(* Logix 5000 project; controller cow Emulate 5570 rev 36.11; software revision 36.00; part 6 of 6 *)
(* tags used below, declared in another part *)
   Batch_delay : TIMER;
   Big_Add : TIMER;
   Big_Avg : REAL;
   Big_Bin_Changed : BOOL;
   Big_Bridge_time : TIMER;
   Big_Error_Over : BOOL;
   Big_ErrorWeight : REAL;
   Big_id : DINT;
   Big_id1 : DINT;
   Big_Idx : DINT;
   Big_Index : DINT;
   Big_Run_Fs : BOOL;
   Big_Scale1 : REAL;
   Big_Scale2 : REAL;
   Big_Scale3 : REAL;
   Big_Timer : TIMER;
   BigBin_Change_ID : DINT;
   Bin_Index : DINT;
   Find : BOOL;
   Hand_Index : DINT;
   Hand_Scale1 : REAL;
   Index : DINT;
   INDEX1 : DINT;
   Max_BigID : DINT;
   No_Big_CMD : BOOL;
   Ons : BOOL[64];
   Part_Index : DINT;
   rcp_Big1 : Part_Type;
   rcp_Big_Bridge_delay : TIMER;
   rcp_BigBin_Bridge : DINT;
   rcp_BigLastID1 : DINT;
   Recipe_Mult : CONTROL;
   Report_TIMER : TIMER;
   Scale_Simulate_Timer : TIMER;
   Simulate_Big_w : REAL;
   ZERO : DINT[100];
   Bin01 : ALIAS FOR rcp_Big_Bin[0];
   Bin02 : ALIAS FOR rcp_Big_Bin[1];
   Bin03 : ALIAS FOR rcp_Big_Bin[2];
   Bin04 : ALIAS FOR rcp_Big_Bin[3];
   Bin05 : ALIAS FOR rcp_Big_Bin[4];
   Bin06 : ALIAS FOR rcp_Big_Bin[5];
   Bin07 : ALIAS FOR rcp_Big_Bin[6];
   Bin08 : ALIAS FOR rcp_Big_Bin[7];
   Bin09 : ALIAS FOR rcp_Big_Bin[8];
   Bin10 : ALIAS FOR rcp_Big_Bin[9];
   Bin11 : ALIAS FOR rcp_Big_Bin[10];
   Bin12 : ALIAS FOR rcp_Big_Bin[11];
   Bin13 : ALIAS FOR rcp_Big_Bin[12];
   Bin14 : ALIAS FOR rcp_Big_Bin[13];
   Bin15 : ALIAS FOR rcp_Big_Bin[14];
   Bin16 : ALIAS FOR rcp_Big_Bin[15];
   E331 : SCALE_WEIGHT;
   E351 : Valve;
   E352 : Valve;
   LED_Batch_seq : DINT;
   LED_Batch_Total : ALIAS FOR rcp_Recipe.BatchSet;
   Led_Hand_PartNumber : DINT;
   Led_Hand_RealWeight : REAL;
   LED_Hand_SetWeight : REAL;
   Now : DateTime_Type;
   rcp_Auto : ALIAS FOR SYS_E.AUTO;
   rcp_Batch : DINT;
   rcp_Batch_OK : BOOL;
   rcp_Batch_Start : BOOL;
   rcp_Big : Part_Type;
   rcp_Big_Add : BOOL;
   rcp_Big_Add_Cmd : BOOL;
   rcp_Big_Add_Skip : BOOL;
   rcp_Big_Bin : Bin_Raw[20];
   rcp_Big_Bridge : BOOL;
   rcp_Big_Bridge_skip : BOOL;
   rcp_Big_Continue : BOOL;
   rcp_Big_Pause : BOOL;
   rcp_Big_Run : BOOL;
   rcp_Big_Scale : REAL;
   rcp_Big_Speed : DINT;
   rcp_BigBin_Change : DINT;
   rcp_BigLastID : DINT;
   rcp_Cancel_Pause : BOOL;
   rcp_class : DINT;
   rcp_Clear : BOOL;
   rcp_Dest_Bin : DINT;
   rcp_Hand : Part_Type_Hand;
   rcp_Hand_Index : DINT;
   rcp_Hand_PB : BOOL;
   rcp_Hand_Run : BOOL;
   rcp_Hand_Scale : REAL;
   rcp_Hand_Total : DINT;
   rcp_Mult : REAL;
   rcp_Recipe : Recipe_Type;
   rcp_Recipe_pNumber : DINT[20];
   rcp_Recipe_Power_Reset : BOOL;
   rcp_Recipe_pSetweight : REAL[20];
   rcp_Recipe_Reset : BOOL;
   rcp_Report_Bin : INT[66];
   rcp_Report_Log : BOOL;
   rcp_Report_Number : DINT[60];
   rcp_Report_RealWeight : REAL[60];
   rcp_Report_SetWeight : REAL[60];
   rcp_RUN : BOOL;
   rcp_Scale_Lock : BOOL;
   rcp_schedule : Recipe_Type[11];
   rcp_schedule_Index : DINT;
   rcp_Schedule_INPUT : BOOL;
   rcp_ScheduleLog : ScheduleLog[10];
   rcp_Set_Pause : BOOL;
   SCALE_SIMULATE : BOOL;
   SYS : System_Common;
(* Recipe, continued *)

ROUTINE MainRoutine   (* ladder *)
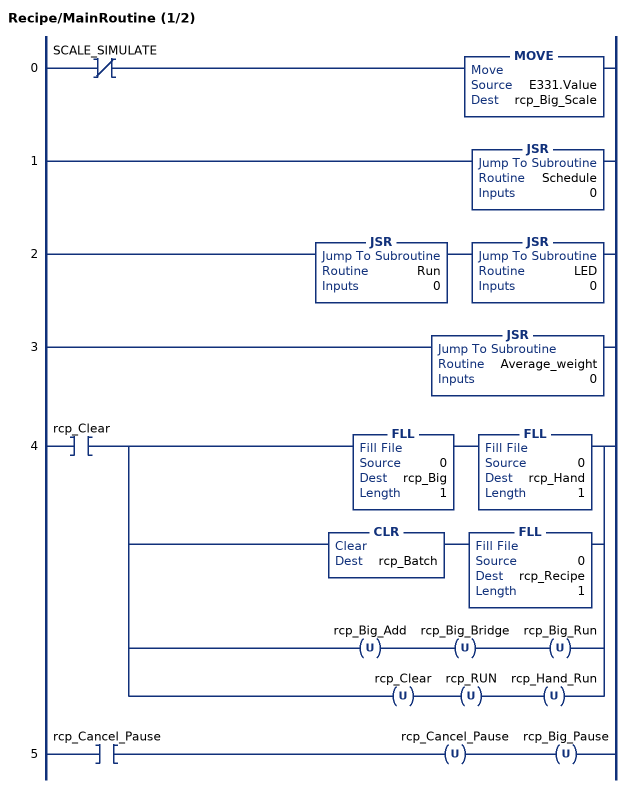
   0: XIO(SCALE_SIMULATE)MOVE(E331.Value,rcp_Big_Scale);
   1: JSR(Schedule,0);
   2: JSR(Run,0)JSR(LED,0);
   3: JSR(Average_weight,0);
   4: XIC(rcp_Clear)[FLL(0,rcp_Big,1) FLL(0,rcp_Hand,1) ,CLR(rcp_Batch) FLL(0,rcp_Recipe,1) ,OTU(rcp_Big_Add) OTU(rcp_Big_Bridge) OTU(rcp_Big_Run) ,OTU(rcp_Clear) OTU(rcp_RUN) OTU(rcp_Hand_Run) ];
   5: XIC(rcp_Cancel_Pause)OTU(rcp_Cancel_Pause)OTU(rcp_Big_Pause);
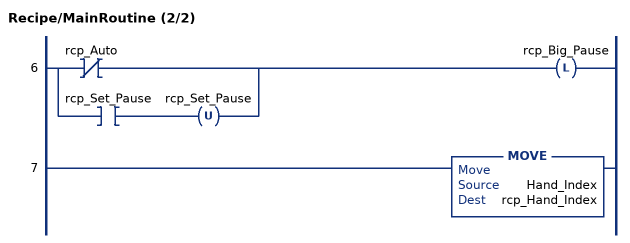
   6: [XIO(rcp_Auto) ,XIC(rcp_Set_Pause) OTU(rcp_Set_Pause) ]OTL(rcp_Big_Pause);
   7: MOVE(Hand_Index,rcp_Hand_Index);
END_ROUTINE

ROUTINE Run   (* ladder *)
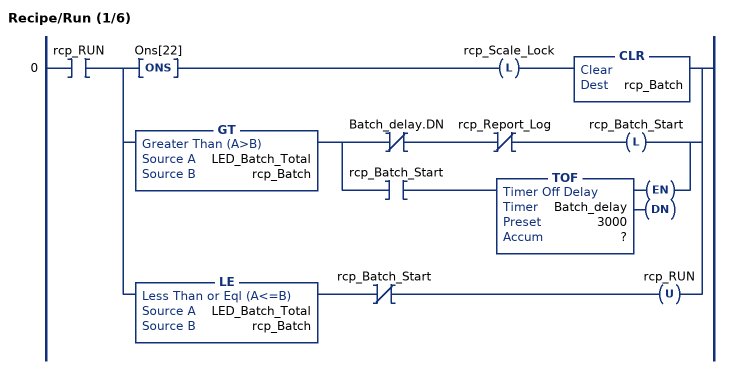
   0: XIC(rcp_RUN)[ONS(Ons[22]) OTL(rcp_Scale_Lock) CLR(rcp_Batch) ,GT(LED_Batch_Total,rcp_Batch) [XIO(Batch_delay.DN) XIO(rcp_Report_Log) OTL(rcp_Batch_Start) ,XIC(rcp_Batch_Start) TOF(Batch_delay,?,?) ] ,LE(LED_Batch_Total,rcp_Batch) XIO(rcp_Batch_Start) OTU(rcp_RUN) ];
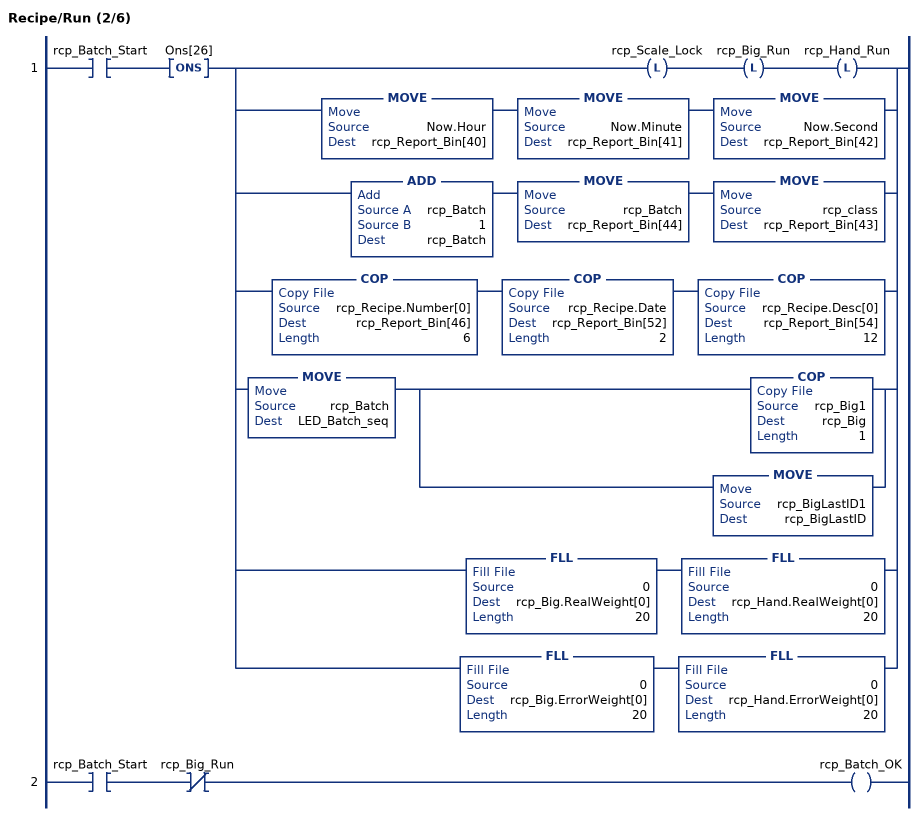
   1: XIC(rcp_Batch_Start)ONS(Ons[26])[OTL(rcp_Scale_Lock) OTL(rcp_Big_Run) OTL(rcp_Hand_Run) ,MOVE(Now.Hour,rcp_Report_Bin[40]) MOVE(Now.Minute,rcp_Report_Bin[41]) MOVE(Now.Second,rcp_Report_Bin[42]) ,ADD(rcp_Batch,1,rcp_Batch) MOVE(rcp_Batch,rcp_Report_Bin[44]) MOVE(rcp_class,rcp_Report_Bin[43]) ,COP(rcp_Recipe.Number[0],rcp_Report_Bin[46],6) COP(rcp_Recipe.Date,rcp_Report_Bin[52],2) COP(rcp_Recipe.Desc[0],rcp_Report_Bin[54],12) ,MOVE(rcp_Batch,LED_Batch_seq) [COP(rcp_Big1,rcp_Big,1) ,MOVE(rcp_BigLastID1,rcp_BigLastID) ] ,FLL(0,rcp_Big.RealWeight[0],20) FLL(0,rcp_Hand.RealWeight[0],20) ,FLL(0,rcp_Big.ErrorWeight[0],20) FLL(0,rcp_Hand.ErrorWeight[0],20) ];
   2: XIC(rcp_Batch_Start)XIO(rcp_Big_Run)OTE(rcp_Batch_OK);
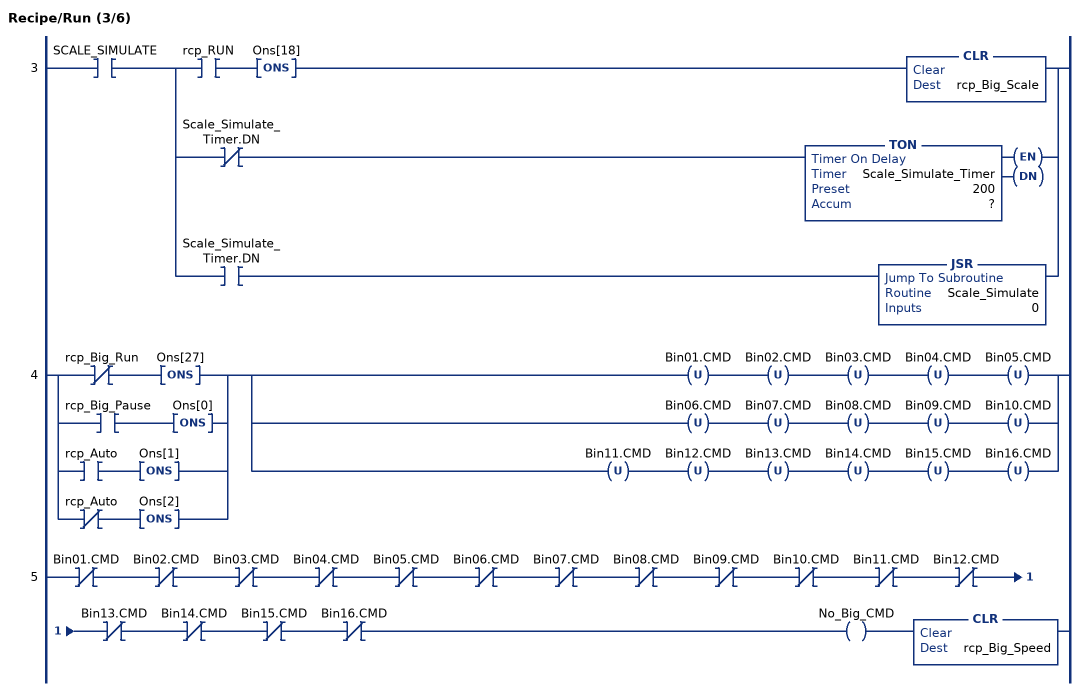
   3: XIC(SCALE_SIMULATE)[XIC(rcp_RUN) ONS(Ons[18]) CLR(rcp_Big_Scale) ,XIO(Scale_Simulate_Timer.DN) TON(Scale_Simulate_Timer,?,?) ,XIC(Scale_Simulate_Timer.DN) JSR(Scale_Simulate,0) ];
   4: [XIO(rcp_Big_Run) ONS(Ons[27]) ,XIC(rcp_Big_Pause) ONS(Ons[0]) ,XIC(rcp_Auto) ONS(Ons[1]) ,XIO(rcp_Auto) ONS(Ons[2]) ][OTU(Bin01.CMD) OTU(Bin02.CMD) OTU(Bin03.CMD) OTU(Bin04.CMD) OTU(Bin05.CMD) ,OTU(Bin06.CMD) OTU(Bin07.CMD) OTU(Bin08.CMD) OTU(Bin09.CMD) OTU(Bin10.CMD) ,OTU(Bin11.CMD) OTU(Bin12.CMD) OTU(Bin13.CMD) OTU(Bin14.CMD) OTU(Bin15.CMD) OTU(Bin16.CMD) ];
   5: XIO(Bin01.CMD)XIO(Bin02.CMD)XIO(Bin03.CMD)XIO(Bin04.CMD)XIO(Bin05.CMD)XIO(Bin06.CMD)XIO(Bin07.CMD)XIO(Bin08.CMD)XIO(Bin09.CMD)XIO(Bin10.CMD)XIO(Bin11.CMD)XIO(Bin12.CMD)XIO(Bin13.CMD)XIO(Bin14.CMD)XIO(Bin15.CMD)XIO(Bin16.CMD)OTE(No_Big_CMD)CLR(rcp_Big_Speed);
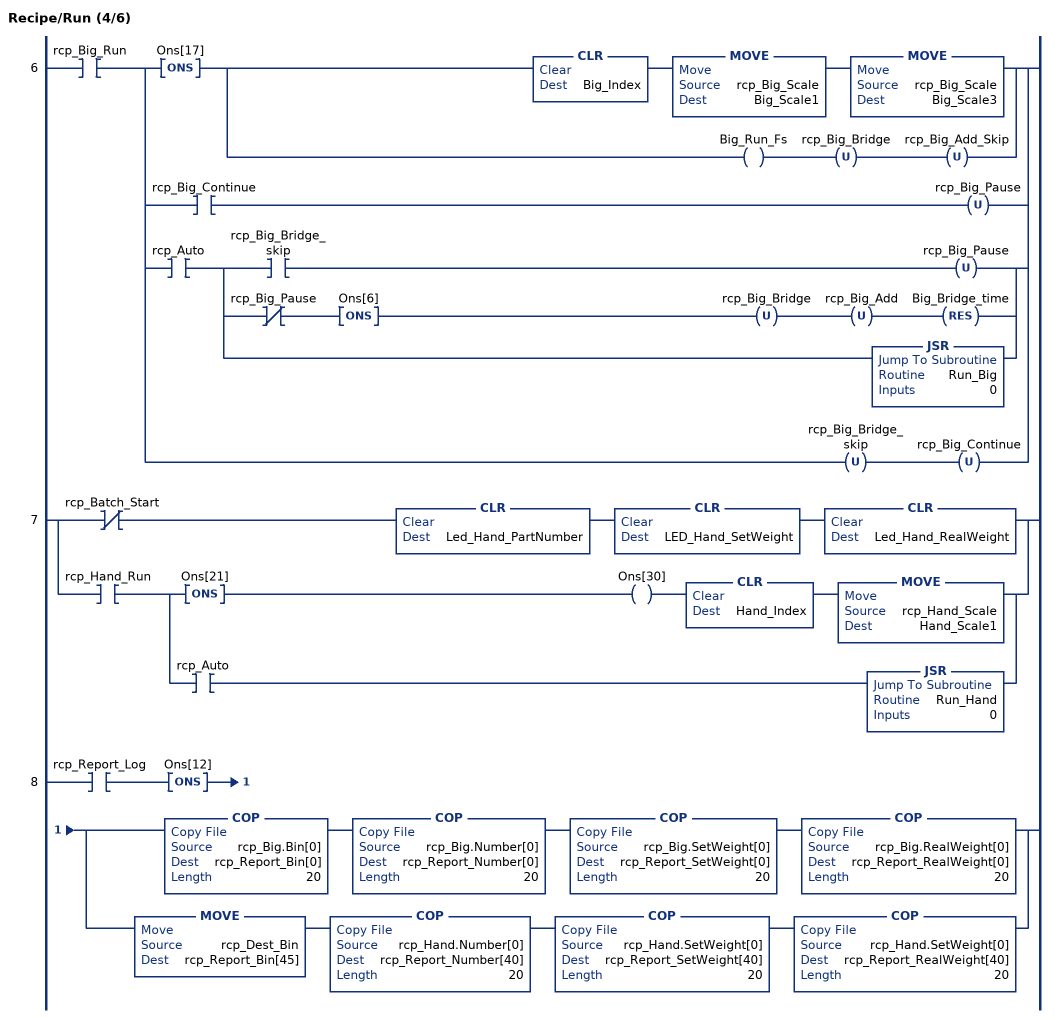
   6: XIC(rcp_Big_Run)[ONS(Ons[17]) [CLR(Big_Index) MOVE(rcp_Big_Scale,Big_Scale1) MOVE(rcp_Big_Scale,Big_Scale3) ,OTE(Big_Run_Fs) OTU(rcp_Big_Bridge) OTU(rcp_Big_Add_Skip) ] ,XIC(rcp_Big_Continue) OTU(rcp_Big_Pause) ,XIC(rcp_Auto) [XIC(rcp_Big_Bridge_skip) OTU(rcp_Big_Pause) ,[XIO(rcp_Big_Pause) ONS(Ons[6]) OTU(rcp_Big_Bridge) OTU(rcp_Big_Add) RES(Big_Bridge_time) ,JSR(Run_Big,0) ] ] ,OTU(rcp_Big_Bridge_skip) OTU(rcp_Big_Continue) ];
   7: [XIO(rcp_Batch_Start) CLR(Led_Hand_PartNumber) CLR(LED_Hand_SetWeight) CLR(Led_Hand_RealWeight) ,XIC(rcp_Hand_Run) [ONS(Ons[21]) OTE(Ons[30]) CLR(Hand_Index) MOVE(rcp_Hand_Scale,Hand_Scale1) ,XIC(rcp_Auto) JSR(Run_Hand,0) ] ];
   8: XIC(rcp_Report_Log)ONS(Ons[12])[COP(rcp_Big.Bin[0],rcp_Report_Bin[0],20) COP(rcp_Big.Number[0],rcp_Report_Number[0],20) COP(rcp_Big.SetWeight[0],rcp_Report_SetWeight[0],20) COP(rcp_Big.RealWeight[0],rcp_Report_RealWeight[0],20) ,MOVE(rcp_Dest_Bin,rcp_Report_Bin[45]) COP(rcp_Hand.Number[0],rcp_Report_Number[40],20) COP(rcp_Hand.SetWeight[0],rcp_Report_SetWeight[40],20) COP(rcp_Hand.SetWeight[0],rcp_Report_RealWeight[40],20) ];
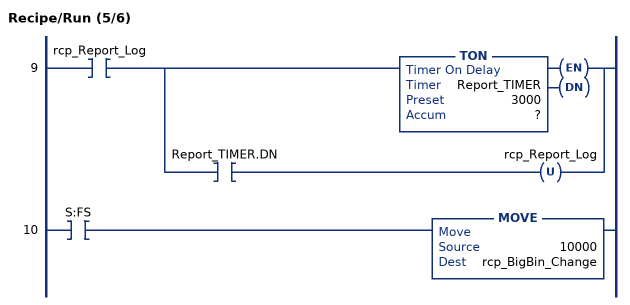
   9: XIC(rcp_Report_Log)[TON(Report_TIMER,?,?) ,XIC(Report_TIMER.DN) OTU(rcp_Report_Log) ];
   10: XIC(S:FS)MOVE(10000,rcp_BigBin_Change);
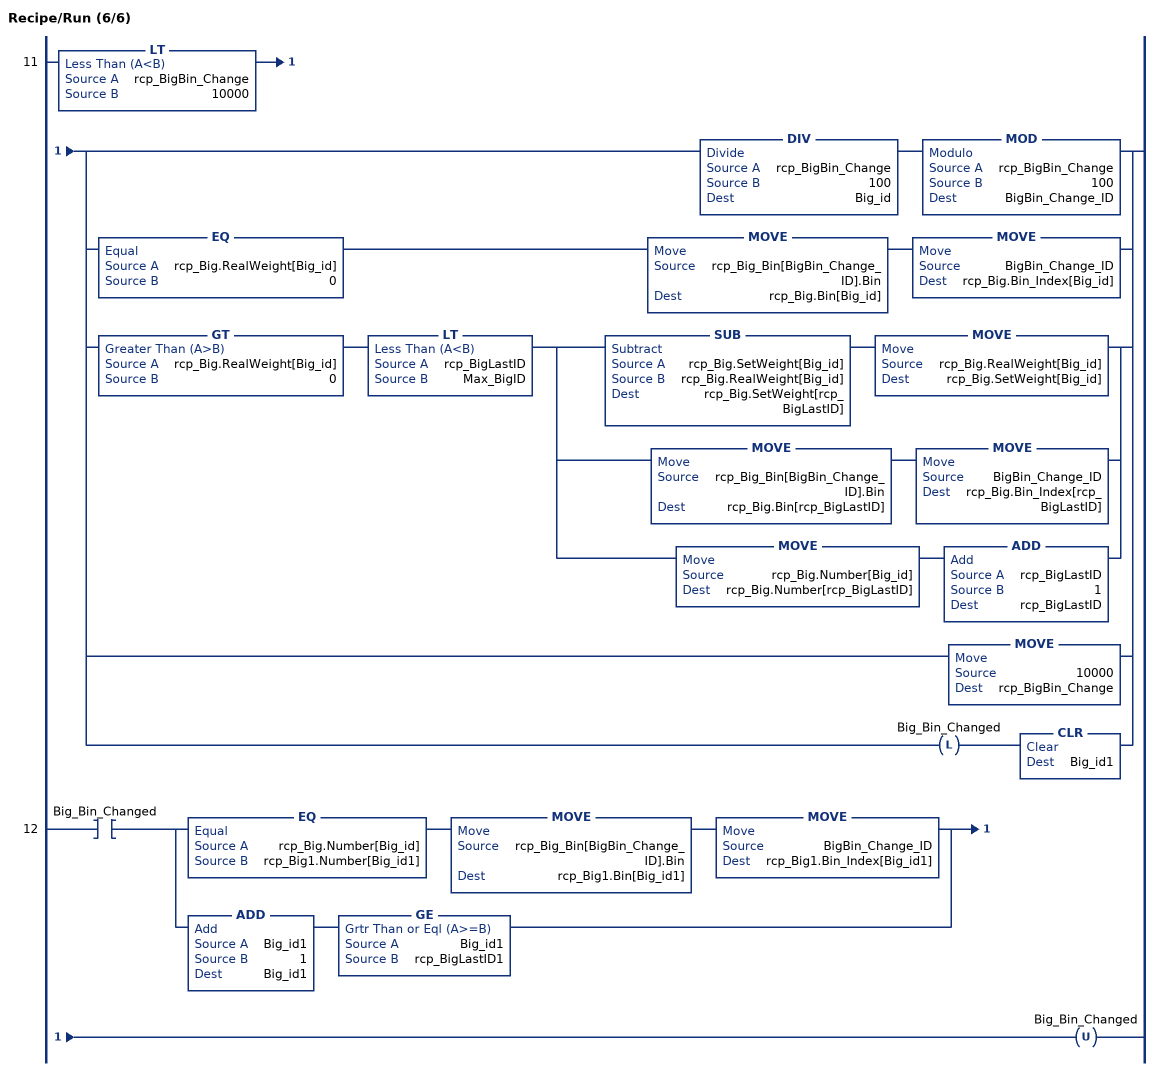
   11: LT(rcp_BigBin_Change,10000)[DIV(rcp_BigBin_Change,100,Big_id) MOD(rcp_BigBin_Change,100,BigBin_Change_ID) ,EQ(rcp_Big.RealWeight[Big_id],0) MOVE(rcp_Big_Bin[BigBin_Change_ID].Bin,rcp_Big.Bin[Big_id]) MOVE(BigBin_Change_ID,rcp_Big.Bin_Index[Big_id]) ,GT(rcp_Big.RealWeight[Big_id],0) LT(rcp_BigLastID,Max_BigID) [SUB(rcp_Big.SetWeight[Big_id],rcp_Big.RealWeight[Big_id],rcp_Big.SetWeight[rcp_BigLastID]) MOVE(rcp_Big.RealWeight[Big_id],rcp_Big.SetWeight[Big_id]) ,MOVE(rcp_Big_Bin[BigBin_Change_ID].Bin,rcp_Big.Bin[rcp_BigLastID]) MOVE(BigBin_Change_ID,rcp_Big.Bin_Index[rcp_BigLastID]) ,MOVE(rcp_Big.Number[Big_id],rcp_Big.Number[rcp_BigLastID]) ADD(rcp_BigLastID,1,rcp_BigLastID) ] ,MOVE(10000,rcp_BigBin_Change) ,OTL(Big_Bin_Changed) CLR(Big_id1) ];
   12: XIC(Big_Bin_Changed)[EQ(rcp_Big.Number[Big_id],rcp_Big1.Number[Big_id1]) MOVE(rcp_Big_Bin[BigBin_Change_ID].Bin,rcp_Big1.Bin[Big_id1]) MOVE(BigBin_Change_ID,rcp_Big1.Bin_Index[Big_id1]) ,ADD(Big_id1,1,Big_id1) GE(Big_id1,rcp_BigLastID1) ]OTU(Big_Bin_Changed);
END_ROUTINE

ROUTINE Run_Big   (* ladder *)
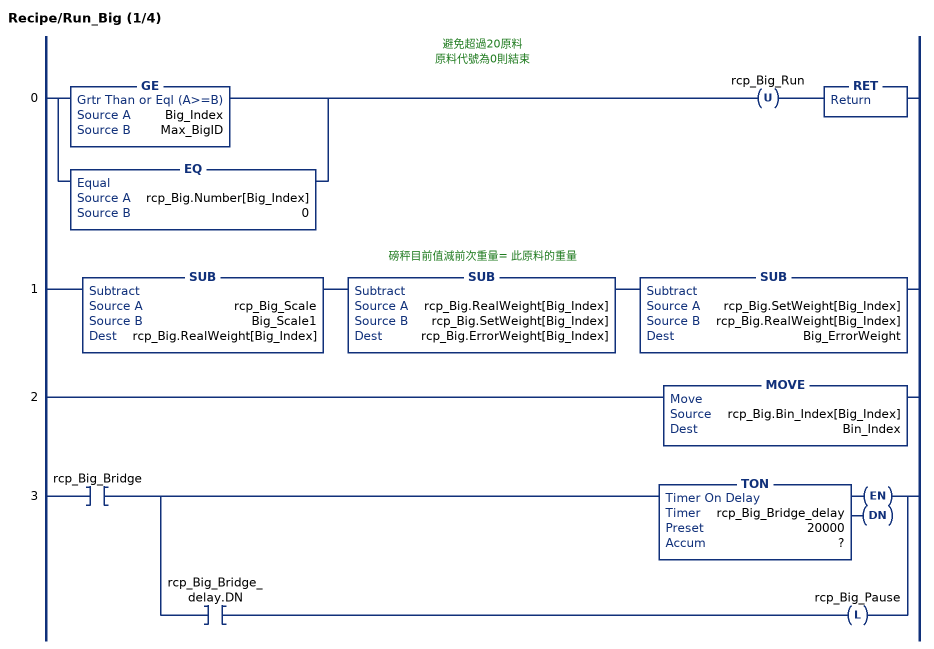
   // 避免超過20原料
   // 原料代號為0則結束
   0: [GE(Big_Index,Max_BigID) ,EQ(rcp_Big.Number[Big_Index],0) ]OTU(rcp_Big_Run)RET();
   // 磅秤目前值減前次重量= 此原料的重量
   1: SUB(rcp_Big_Scale,Big_Scale1,rcp_Big.RealWeight[Big_Index])SUB(rcp_Big.RealWeight[Big_Index],rcp_Big.SetWeight[Big_Index],rcp_Big.ErrorWeight[Big_Index])SUB(rcp_Big.SetWeight[Big_Index],rcp_Big.RealWeight[Big_Index],Big_ErrorWeight);
   2: MOVE(rcp_Big.Bin_Index[Big_Index],Bin_Index);
   3: XIC(rcp_Big_Bridge)[TON(rcp_Big_Bridge_delay,?,?) ,XIC(rcp_Big_Bridge_delay.DN) OTL(rcp_Big_Pause) ];
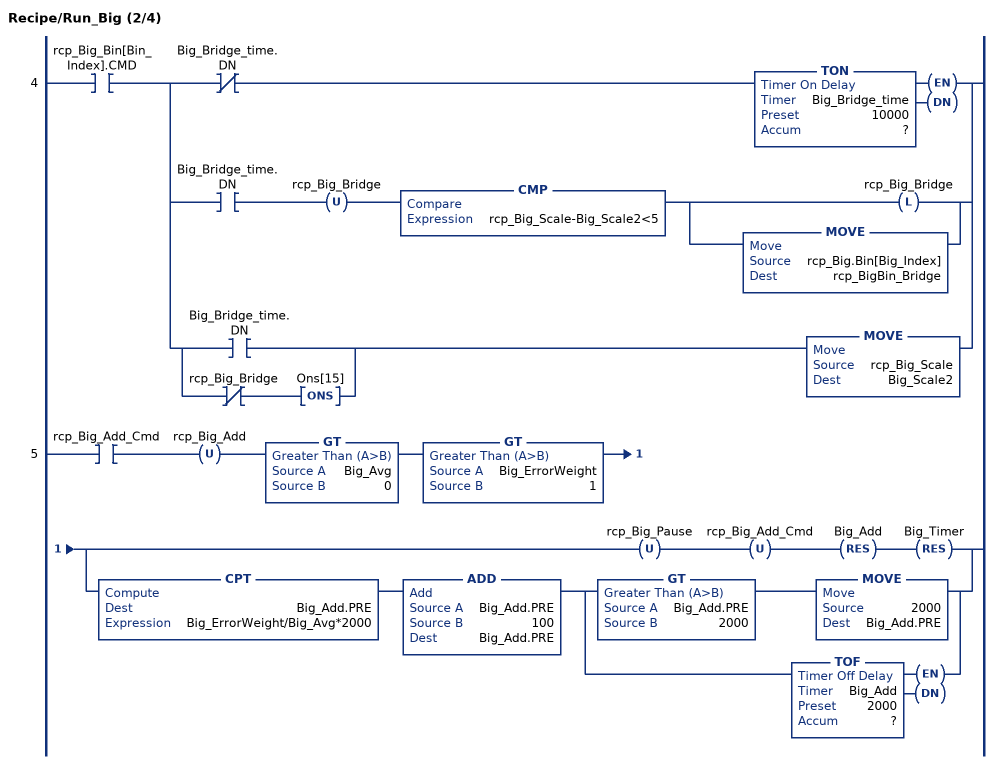
   4: XIC(rcp_Big_Bin[Bin_Index].CMD)[XIO(Big_Bridge_time.DN) TON(Big_Bridge_time,?,?) ,XIC(Big_Bridge_time.DN) OTU(rcp_Big_Bridge) CMP(rcp_Big_Scale-Big_Scale2<5) [OTL(rcp_Big_Bridge) ,MOVE(rcp_Big.Bin[Big_Index],rcp_BigBin_Bridge) ] ,[XIC(Big_Bridge_time.DN) ,XIO(rcp_Big_Bridge) ONS(Ons[15]) ] MOVE(rcp_Big_Scale,Big_Scale2) ];
   5: XIC(rcp_Big_Add_Cmd)OTU(rcp_Big_Add)GT(Big_Avg,0)GT(Big_ErrorWeight,1)[OTU(rcp_Big_Pause) OTU(rcp_Big_Add_Cmd) RES(Big_Add) RES(Big_Timer) ,CPT(Big_Add.PRE,Big_ErrorWeight/Big_Avg*2000) ADD(Big_Add.PRE,100,Big_Add.PRE) [GT(Big_Add.PRE,2000) MOVE(2000,Big_Add.PRE) ,TOF(Big_Add,?,?) ] ];
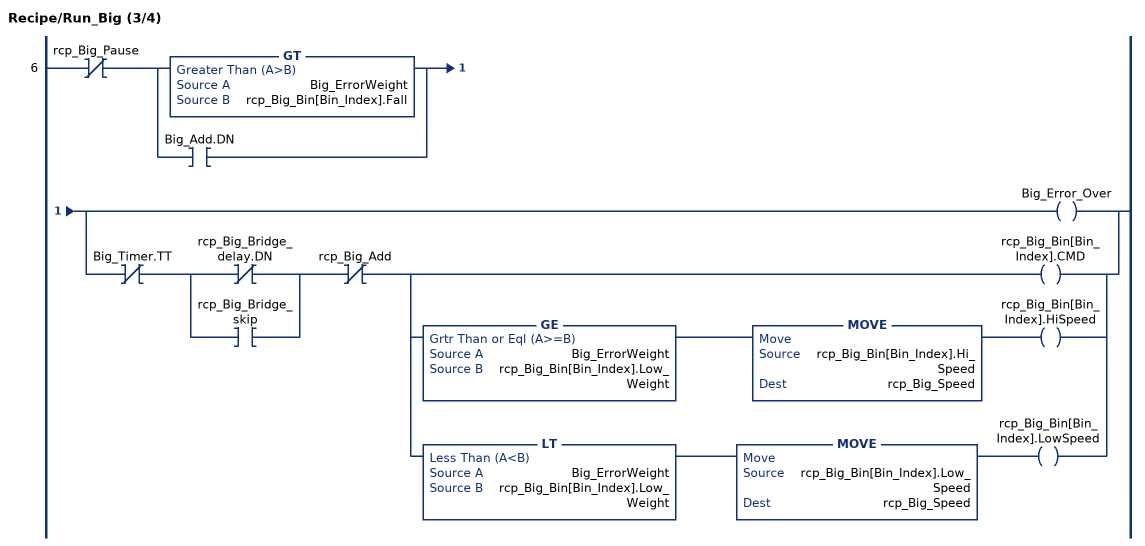
   6: XIO(rcp_Big_Pause)[GT(Big_ErrorWeight,rcp_Big_Bin[Bin_Index].Fall) ,XIC(Big_Add.DN) ][OTE(Big_Error_Over) ,XIO(Big_Timer.TT) [XIO(rcp_Big_Bridge_delay.DN) ,XIC(rcp_Big_Bridge_skip) ] XIO(rcp_Big_Add) [OTE(rcp_Big_Bin[Bin_Index].CMD) ,GE(Big_ErrorWeight,rcp_Big_Bin[Bin_Index].Low_Weight) MOVE(rcp_Big_Bin[Bin_Index].Hi_Speed,rcp_Big_Speed) OTE(rcp_Big_Bin[Bin_Index].HiSpeed) ,LT(Big_ErrorWeight,rcp_Big_Bin[Bin_Index].Low_Weight) MOVE(rcp_Big_Bin[Bin_Index].Low_Speed,rcp_Big_Speed) OTE(rcp_Big_Bin[Bin_Index].LowSpeed) ] ];
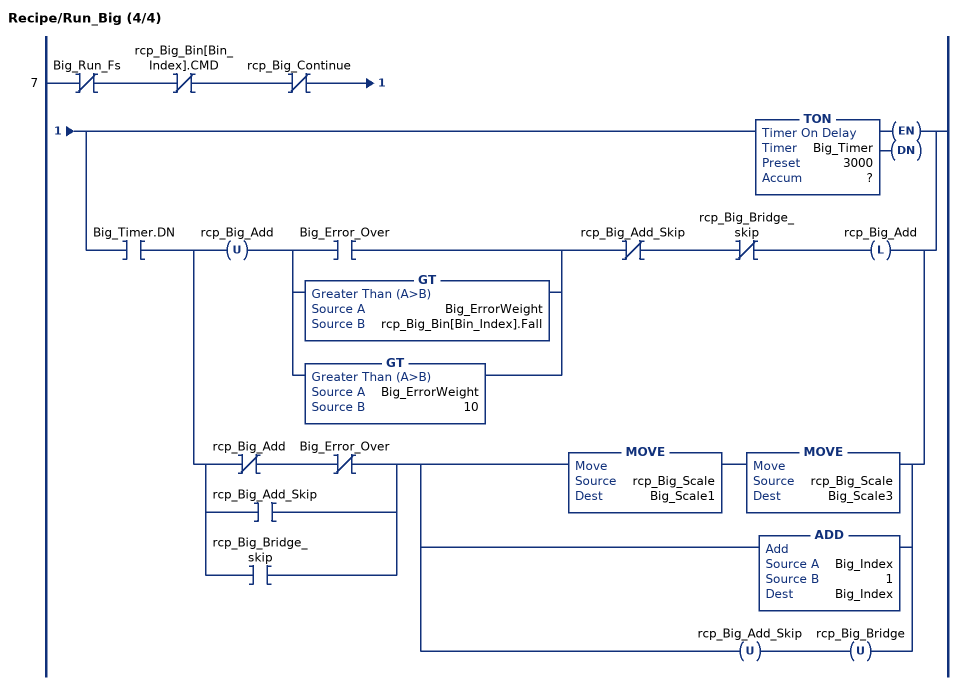
   7: XIO(Big_Run_Fs)XIO(rcp_Big_Bin[Bin_Index].CMD)XIO(rcp_Big_Continue)[TON(Big_Timer,?,?) ,XIC(Big_Timer.DN) [OTU(rcp_Big_Add) [XIC(Big_Error_Over) ,GT(Big_ErrorWeight,rcp_Big_Bin[Bin_Index].Fall) ,GT(Big_ErrorWeight,10) ] XIO(rcp_Big_Add_Skip) XIO(rcp_Big_Bridge_skip) OTL(rcp_Big_Add) ,[XIO(rcp_Big_Add) XIO(Big_Error_Over) ,XIC(rcp_Big_Add_Skip) ,XIC(rcp_Big_Bridge_skip) ] [MOVE(rcp_Big_Scale,Big_Scale1) MOVE(rcp_Big_Scale,Big_Scale3) ,ADD(Big_Index,1,Big_Index) ,OTU(rcp_Big_Add_Skip) OTU(rcp_Big_Bridge) ] ] ];
END_ROUTINE

ROUTINE Run_Hand   (* ladder *)
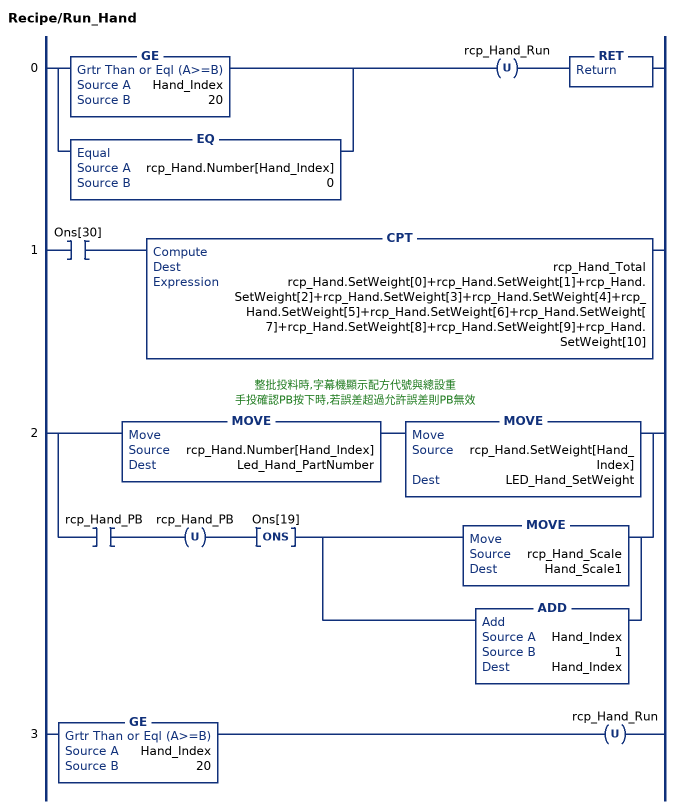
   0: [GE(Hand_Index,20) ,EQ(rcp_Hand.Number[Hand_Index],0) ]OTU(rcp_Hand_Run)RET();
   1: XIC(Ons[30])CPT(rcp_Hand_Total,rcp_Hand.SetWeight[0]+rcp_Hand.SetWeight[1]+rcp_Hand.SetWeight[2]+rcp_Hand.SetWeight[3]+rcp_Hand.SetWeight[4]+rcp_Hand.SetWeight[5]+rcp_Hand.SetWeight[6]+rcp_Hand.SetWeight[7]+rcp_Hand.SetWeight[8]+rcp_Hand.SetWeight[9]+rcp_Hand.SetWeight[10]);
   // 整批投料時,字幕機顯示配方代號與總設重
   // 手投確認PB按下時,若誤差超過允許誤差則PB無效
   2: [MOVE(rcp_Hand.Number[Hand_Index],Led_Hand_PartNumber) MOVE(rcp_Hand.SetWeight[Hand_Index],LED_Hand_SetWeight) ,XIC(rcp_Hand_PB) OTU(rcp_Hand_PB) ONS(Ons[19]) [MOVE(rcp_Hand_Scale,Hand_Scale1) ,ADD(Hand_Index,1,Hand_Index) ] ];
   3: GE(Hand_Index,20)OTU(rcp_Hand_Run);
END_ROUTINE

ROUTINE Scale_Simulate   (* ladder *)
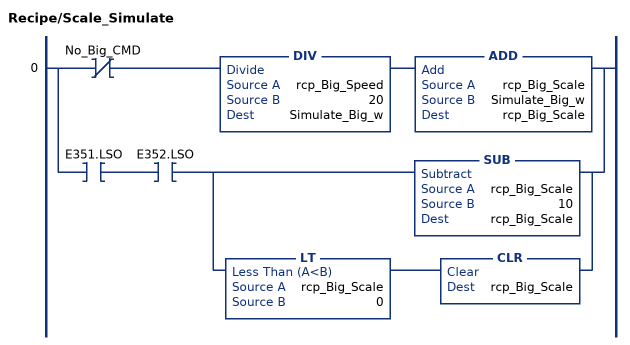
   0: [XIO(No_Big_CMD) DIV(rcp_Big_Speed,20,Simulate_Big_w) ADD(rcp_Big_Scale,Simulate_Big_w,rcp_Big_Scale) ,XIC(E351.LSO) XIC(E352.LSO) [SUB(rcp_Big_Scale,10,rcp_Big_Scale) ,LT(rcp_Big_Scale,0) CLR(rcp_Big_Scale) ] ];
END_ROUTINE

ROUTINE Schedule   (* ladder *)
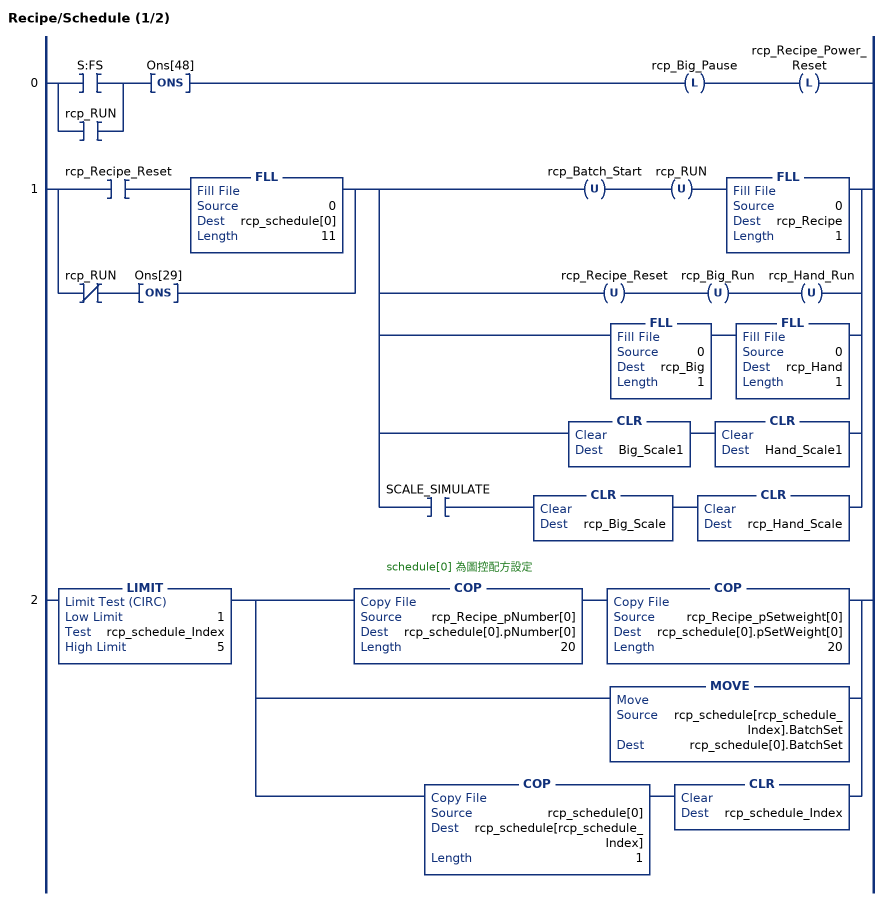
   0: [XIC(S:FS) ,XIC(rcp_RUN) ]ONS(Ons[48])OTL(rcp_Big_Pause)OTL(rcp_Recipe_Power_Reset);
   1: [XIC(rcp_Recipe_Reset) FLL(0,rcp_schedule[0],11) ,XIO(rcp_RUN) ONS(Ons[29]) ][OTU(rcp_Batch_Start) OTU(rcp_RUN) FLL(0,rcp_Recipe,1) ,OTU(rcp_Recipe_Reset) OTU(rcp_Big_Run) OTU(rcp_Hand_Run) ,FLL(0,rcp_Big,1) FLL(0,rcp_Hand,1) ,CLR(Big_Scale1) CLR(Hand_Scale1) ,XIC(SCALE_SIMULATE) CLR(rcp_Big_Scale) CLR(rcp_Hand_Scale) ];
   // schedule[0] 為圖控配方設定
   2: LIMIT(1,rcp_schedule_Index,5)[COP(rcp_Recipe_pNumber[0],rcp_schedule[0].pNumber[0],20) COP(rcp_Recipe_pSetweight[0],rcp_schedule[0].pSetWeight[0],20) ,MOVE(rcp_schedule[rcp_schedule_Index].BatchSet,rcp_schedule[0].BatchSet) ,COP(rcp_schedule[0],rcp_schedule[rcp_schedule_Index],1) CLR(rcp_schedule_Index) ];
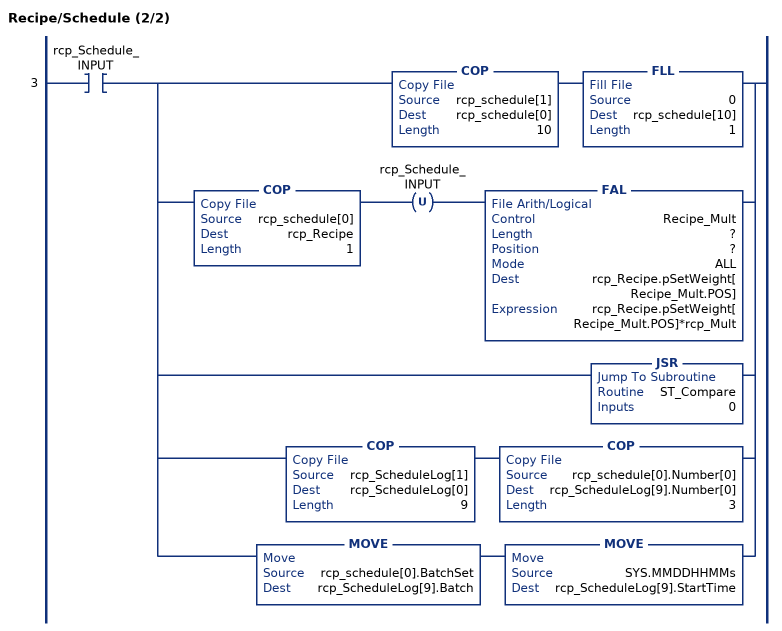
   3: XIC(rcp_Schedule_INPUT)[COP(rcp_schedule[1],rcp_schedule[0],10) FLL(0,rcp_schedule[10],1) ,COP(rcp_schedule[0],rcp_Recipe,1) OTU(rcp_Schedule_INPUT) FAL(Recipe_Mult,?,?,ALL,rcp_Recipe.pSetWeight[Recipe_Mult.POS],rcp_Recipe.pSetWeight[Recipe_Mult.POS]*rcp_Mult) ,JSR(ST_Compare,0) ,COP(rcp_ScheduleLog[1],rcp_ScheduleLog[0],9) COP(rcp_schedule[0].Number[0],rcp_ScheduleLog[9].Number[0],3) ,MOVE(rcp_schedule[0].BatchSet,rcp_ScheduleLog[9].Batch) MOVE(SYS.MMDDHHMMs,rcp_ScheduleLog[9].StartTime) ];
END_ROUTINE

ROUTINE ST_Compare   (* structured text *)
   COP(ZERO[0],rcp_Big,1);COP(ZERO[0],rcp_Hand,1);
   Big_Idx:=0;Hand_Index:=0;rcp_Batch:=0;
   FOR Part_Index:= 0 to 19 DO
   IF rcp_Recipe.pNumber[Part_Index]<> 0 THEN
     Find:= 0;   FOR INDEX1:=0 TO 15 DO //Compare Big Bin
          IF Now.Day.0 THEN Index:= INDEX1; ELSE  Index:= 15 -INDEX1;  End_IF;  //單雙日順序
    IF NOT rcp_Big_Bin[Index].Disable & (rcp_Big_Bin[Index].Number= rcp_Recipe.pNumber[Part_Index]) THEN
   	  Find:=1; rcp_Big.Bin[Big_Idx]:= rcp_Big_Bin[Index].Bin ; rcp_Big.Bin_Index[Big_Idx]:= Index;
   	  rcp_Big.Number[Big_Idx]:= rcp_Recipe.pNumber[Part_Index];
   	  rcp_Big.SetWeight[Big_Idx] := rcp_Recipe.pSetWeight[Part_Index];
   	  Big_Idx:= Big_Idx +1;Exit;
   	 End_IF;  End_FOR;
   
      IF NOT Find then //手投
      rcp_Hand.Number[Hand_Index]:= rcp_Recipe.pNumber[Part_Index];  rcp_Hand.SetWeight[Hand_Index]:= rcp_Recipe.pSetWeight[Part_Index];
      IF Hand_Index<19 THEN Hand_Index:=Hand_Index+1;End_IF;
      End_IF;
   
   End_IF; End_FOR;
   rcp_BigLastID:= Big_Idx;
   COP(rcp_Big,rcp_Big1, 1); rcp_BigLastID1:= rcp_BigLastID;
   
END_ROUTINE
END_PROGRAM
